Staubli VAL3: GenericEnc.dtx

public aio aiEncCurrentPos
aio aiEncLatchedPos
aio aoEncResolution
aio aoPresetPos
bool bCountOvf
bool bCountUdf
public bool bLatchEnabled
bool bLatchLevel
bool bMemoLatchState
bool bPartLatched
bool bReset
dio diEncLatched
dio diOverFlow
dio diUnderFlow
dio diLatchSignal
dio doEnableLatch
dio doEnablePreset
dio doResetErr
num nEncValue
num nEncLatchedVal
num nEncResolution = 2000
public num nLatchPeriod = 1
num nPresetPos
string sEncNum
string sTASK = "encoder"
public num nMAXCOUNT
public num nMINCOUNT
